FUNCTION_BLOCK FB_Actuator_TestWithoutTimeDecorator EXTENDS FB_Actuator_TestDecorator
VAR

END_VAR

(*			
	EVERDE sp. z o.o.
	Rafał Osajda		27.03.2025		TC 4024.66
	Wywolanie co cykl operacji 
*)
METHOD PUBLIC ExecuteEveryCycle_Operation
VAR_INPUT
END_VAR
//testować czy jest cykl przesuwania do gdzieś i po czasie uruchamiać lub wyłączać czujniki 
THIS^.itfactActuator.ExecuteEveryCycle_Operation ();

IF (THIS^.itfactActuator.MovingToStartFirstCycle ()) THEN
	THIS^.itfczStart		:= THIS^.itfsenEnd;
	THIS^.itfczStop			:= THIS^.itfsenStart;
	THIS^.iStepTestCycle	:= 10;
END_IF

IF (THIS^.itfactActuator.MovingToEndFirstCycyle ()) THEN
	THIS^.itfczStart		:= THIS^.itfsenStart;
	THIS^.itfczStop			:= THIS^.itfsenEnd;
	THIS^.iStepTestCycle	:= 10;
END_IF

CASE THIS^.iStepTestCycle OF
10	: THIS^.iStepTestCycle	:= THIS^.iStepTestCycle + 10;	//pierwszy cykl
20	: THIS^.iStepTestCycle	:= THIS^.iStepTestCycle + 10;
30	: 
	THIS^.itfczStart.SetContact (bIN := FALSE); 
	THIS^.iStepTestCycle	:= THIS^.iStepTestCycle + 10;
40	: 
	THIS^.itfczStop.SetContact (bIN := TRUE);
	THIS^.iStepTestCycle	:= 0;
END_CASE
END_METHOD

END_FUNCTION_BLOCK

(* stored: Version 1.1.0.1
   POU FB_Actuator_TestWithoutTimeDecorator: Id {d6f6e8b8-31a0-0da4-0040-d419cd3616d4}, SpecialFunc None
   Method ExecuteEveryCycle_Operation: Id {a0022e83-1441-0473-29eb-3c64758fe0e7} *)
